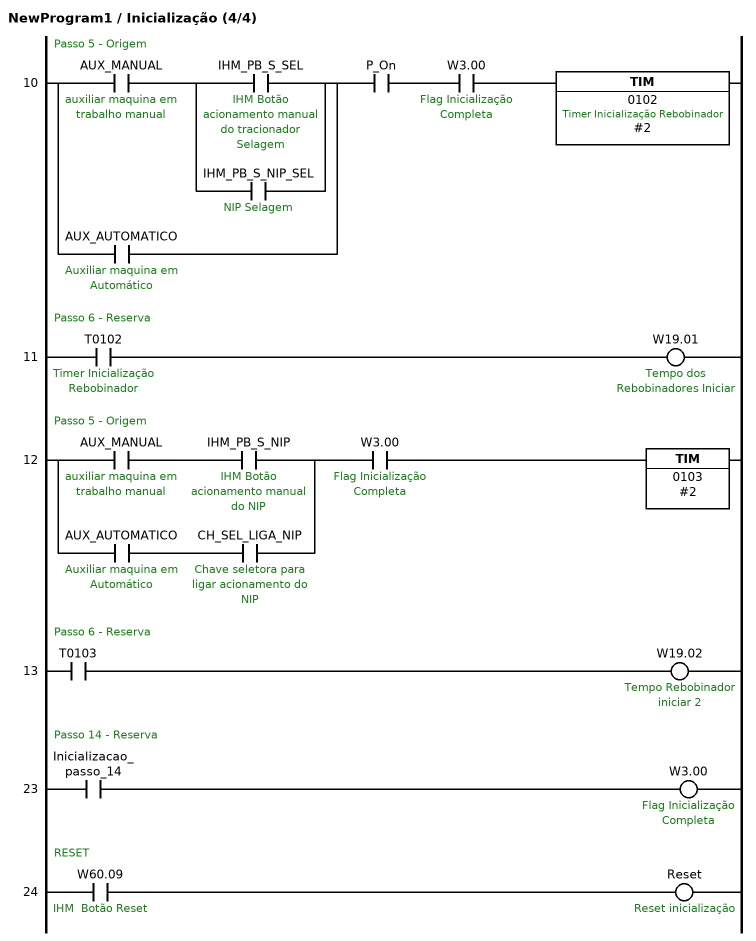
; [picture p24: NewProgram1 / Inicialização, rungs 10-24]
; rung 10: Passo 5 - Origem
LD AUX_MANUAL  ; auxiliar maquina em trabalho manual
LD IHM_PB_S_SEL  ; IHM Botão acionamento manual do tracionador Selagem
OR IHM_PB_S_NIP_SEL  ; NIP Selagem
ANDLD
OR AUX_AUTOMATICO  ; Auxiliar maquina em Automático
AND P_On
AND W3.00  ; Flag Inicialização Completa
TIM 0102 #2  ; Timer Inicialização Rebobinador
; rung 11: Passo 6 - Reserva
LD T0102  ; Timer Inicialização Rebobinador
OUT W19.01  ; Tempo dos Rebobinadores Iniciar
; rung 12: Passo 5 - Origem
LD AUX_MANUAL  ; auxiliar maquina em trabalho manual
AND IHM_PB_S_NIP  ; IHM Botão acionamento manual do NIP
LD AUX_AUTOMATICO  ; Auxiliar maquina em Automático
AND CH_SEL_LIGA_NIP  ; Chave seletora para ligar acionamento do NIP
ORLD
AND W3.00  ; Flag Inicialização Completa
TIM 0103 #2
; rung 13: Passo 6 - Reserva
LD T0103
OUT W19.02  ; Tempo Rebobinador iniciar 2
; rung 14: Passo 5 - Origem
; rung 15: Passo 6 - Reserva
; rung 16: Passo 7 - Reserva
; rung 17: Passo 8 - Reserva
; rung 18: Passo 9 - Reserva
; rung 19: Passo 10 - Reserva
; rung 20: Passo 11 - Reserva
; rung 21: Passo 12 - Reserva
; rung 22: Passo 13 - Reserva
; rung 23: Passo 14 - Reserva
LD Inicializacao_passo_14
OUT W3.00  ; Flag Inicialização Completa
; rung 24: RESET
LD W60.09  ; IHM  Botão Reset
OUT Reset  ; Reset inicialização

### Section Temperatura

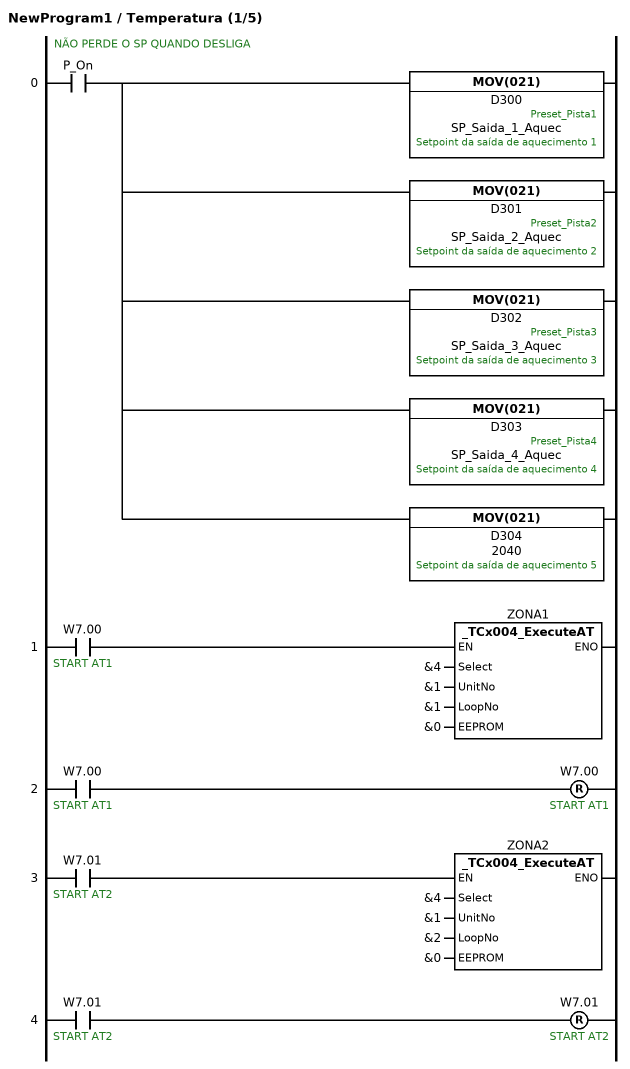
; rung 0: NÃO PERDE O SP QUANDO DESLIGA
LD P_On
MOV(021) D300 SP_Saida_1_Aquec  ; Preset_Pista1, Setpoint da saída de aquecimento 1
MOV(021) D301 SP_Saida_2_Aquec  ; Preset_Pista2, Setpoint da saída de aquecimento 2
MOV(021) D302 SP_Saida_3_Aquec  ; Preset_Pista3, Setpoint da saída de aquecimento 3
MOV(021) D303 SP_Saida_4_Aquec  ; Preset_Pista4, Setpoint da saída de aquecimento 4
MOV(021) D304 2040  ; Setpoint da saída de aquecimento 5
; rung 1
LD W7.00  ; START AT1
CALL ZONA1 : _TCx004_ExecuteAT (Select := &4, UnitNo := &1, LoopNo := &1, EEPROM := &0)
; rung 2
LD W7.00  ; START AT1
RSET W7.00  ; START AT1
; rung 3
LD W7.01  ; START AT2
CALL ZONA2 : _TCx004_ExecuteAT (Select := &4, UnitNo := &1, LoopNo := &2, EEPROM := &0)
; rung 4
LD W7.01  ; START AT2
RSET W7.01  ; START AT2

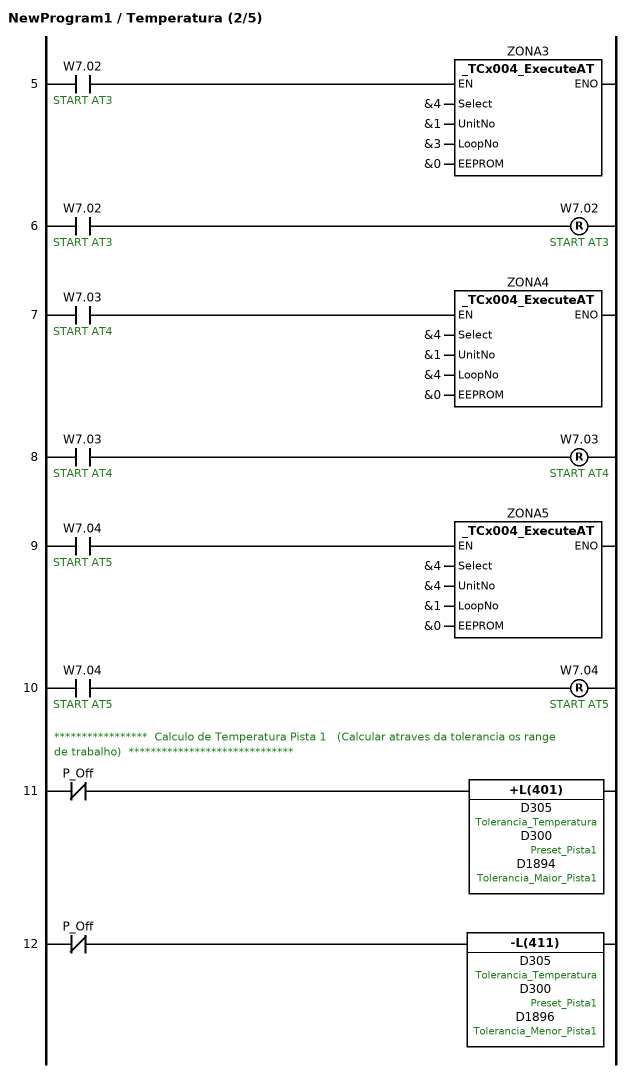
; rung 5
LD W7.02  ; START AT3
CALL ZONA3 : _TCx004_ExecuteAT (Select := &4, UnitNo := &1, LoopNo := &3, EEPROM := &0)
; rung 6
LD W7.02  ; START AT3
RSET W7.02  ; START AT3
; rung 7
LD W7.03  ; START AT4
CALL ZONA4 : _TCx004_ExecuteAT (Select := &4, UnitNo := &1, LoopNo := &4, EEPROM := &0)
; rung 8
LD W7.03  ; START AT4
RSET W7.03  ; START AT4
; rung 9
LD W7.04  ; START AT5
CALL ZONA5 : _TCx004_ExecuteAT (Select := &4, UnitNo := &4, LoopNo := &1, EEPROM := &0)
; rung 10
LD W7.04  ; START AT5
RSET W7.04  ; START AT5
; rung 11: *****************  Calculo de Temperatura Pista 1   (Calcular atraves da tolerancia os range de trabalho)  ******************************
LDNOT P_Off
+L(401) D305 D300 D1894  ; Tolerancia_Temperatura, Preset_Pista1, Tolerancia_Maior_Pista1
; rung 12
LDNOT P_Off
-L(411) D305 D300 D1896  ; Tolerancia_Temperatura, Preset_Pista1, Tolerancia_Menor_Pista1

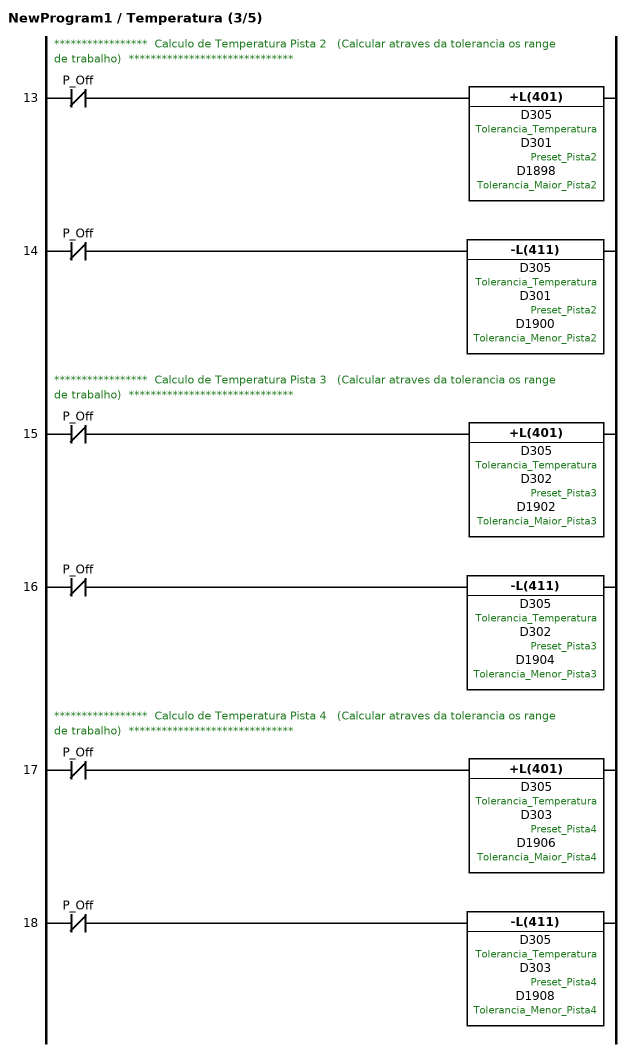
; rung 13: *****************  Calculo de Temperatura Pista 2   (Calcular atraves da tolerancia os range de trabalho)  ******************************
LDNOT P_Off
+L(401) D305 D301 D1898  ; Tolerancia_Temperatura, Preset_Pista2, Tolerancia_Maior_Pista2
; rung 14
LDNOT P_Off
-L(411) D305 D301 D1900  ; Tolerancia_Temperatura, Preset_Pista2, Tolerancia_Menor_Pista2
; rung 15: *****************  Calculo de Temperatura Pista 3   (Calcular atraves da tolerancia os range de trabalho)  ******************************
LDNOT P_Off
+L(401) D305 D302 D1902  ; Tolerancia_Temperatura, Preset_Pista3, Tolerancia_Maior_Pista3
; rung 16
LDNOT P_Off
-L(411) D305 D302 D1904  ; Tolerancia_Temperatura, Preset_Pista3, Tolerancia_Menor_Pista3
; rung 17: *****************  Calculo de Temperatura Pista 4   (Calcular atraves da tolerancia os range de trabalho)  ******************************
LDNOT P_Off
+L(401) D305 D303 D1906  ; Tolerancia_Temperatura, Preset_Pista4, Tolerancia_Maior_Pista4
; rung 18
LDNOT P_Off
-L(411) D305 D303 D1908  ; Tolerancia_Temperatura, Preset_Pista4, Tolerancia_Menor_Pista4

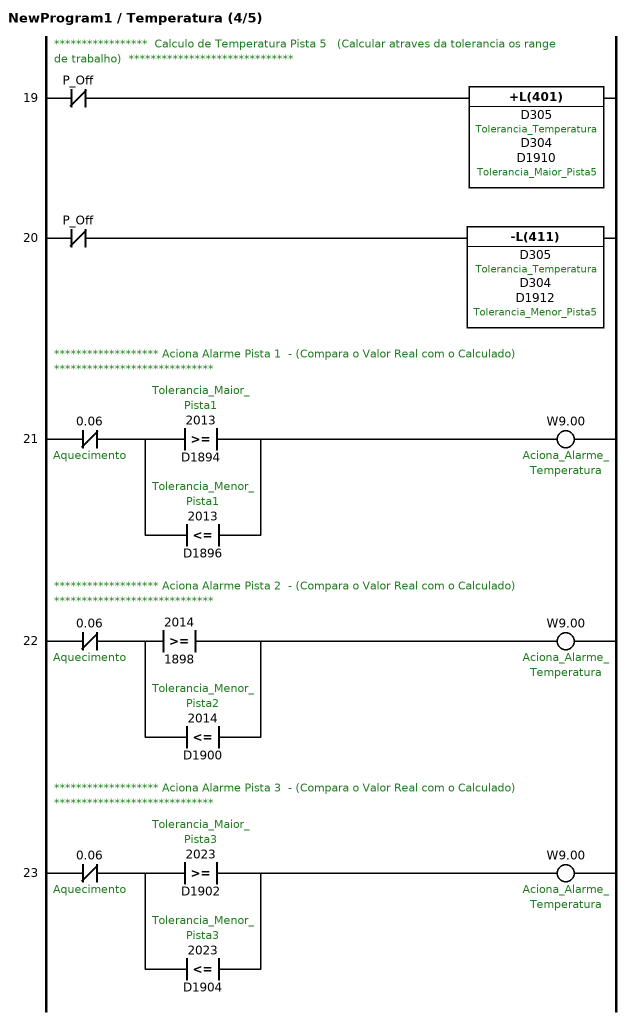
; rung 19: *****************  Calculo de Temperatura Pista 5   (Calcular atraves da tolerancia os range de trabalho)  ******************************
LDNOT P_Off
+L(401) D305 D304 D1910  ; Tolerancia_Temperatura, Tolerancia_Maior_Pista5
; rung 20
LDNOT P_Off
-L(411) D305 D304 D1912  ; Tolerancia_Temperatura, Tolerancia_Menor_Pista5
; rung 21: ******************* Aciona Alarme Pista 1  - (Compara o Valor Real com o Calculado) *****************************
LDNOT 0.06  ; Aquecimento
LD>=L(326) 2013 D1894  ; Tolerancia_Maior_Pista1
OR<=L(316) 2013 D1896  ; Tolerancia_Menor_Pista1
ANDLD
OUT W9.00  ; Aciona_Alarme_Temperatura
; rung 22: ******************* Aciona Alarme Pista 2  - (Compara o Valor Real com o Calculado) *****************************
LDNOT 0.06  ; Aquecimento
LD>=L(326) 2014 1898
OR<=L(316) 2014 D1900  ; Tolerancia_Menor_Pista2
ANDLD
OUT W9.00  ; Aciona_Alarme_Temperatura
; rung 23: ******************* Aciona Alarme Pista 3  - (Compara o Valor Real com o Calculado) *****************************
LDNOT 0.06  ; Aquecimento
LD>=L(326) 2023 D1902  ; Tolerancia_Maior_Pista3
OR<=L(316) 2023 D1904  ; Tolerancia_Menor_Pista3
ANDLD
OUT W9.00  ; Aciona_Alarme_Temperatura

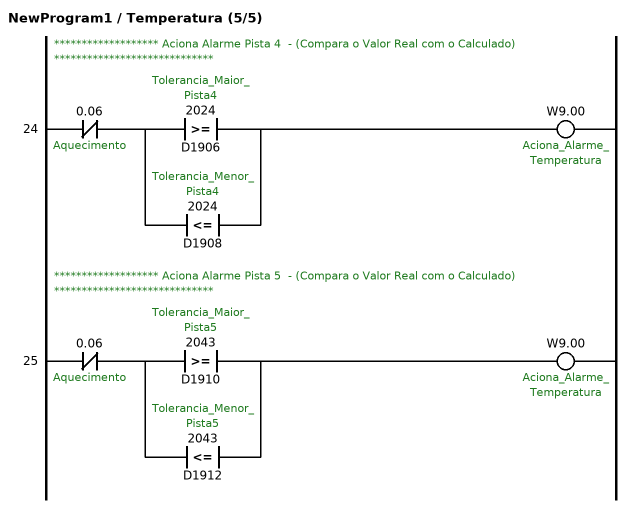
; rung 24: ******************* Aciona Alarme Pista 4  - (Compara o Valor Real com o Calculado) *****************************
LDNOT 0.06  ; Aquecimento
LD>=L(326) 2024 D1906  ; Tolerancia_Maior_Pista4
OR<=L(316) 2024 D1908  ; Tolerancia_Menor_Pista4
ANDLD
OUT W9.00  ; Aciona_Alarme_Temperatura
; rung 25: ******************* Aciona Alarme Pista 5  - (Compara o Valor Real com o Calculado) *****************************
LDNOT 0.06  ; Aquecimento
LD>=L(326) 2043 D1910  ; Tolerancia_Maior_Pista5
OR<=L(316) 2043 D1912  ; Tolerancia_Menor_Pista5
ANDLD
OUT W9.00  ; Aciona_Alarme_Temperatura

### Section Automático

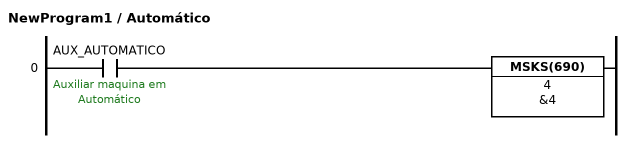
; rung 0
LD AUX_AUTOMATICO  ; Auxiliar maquina em Automático
MSKS(690) 4 &4

### Section Producao

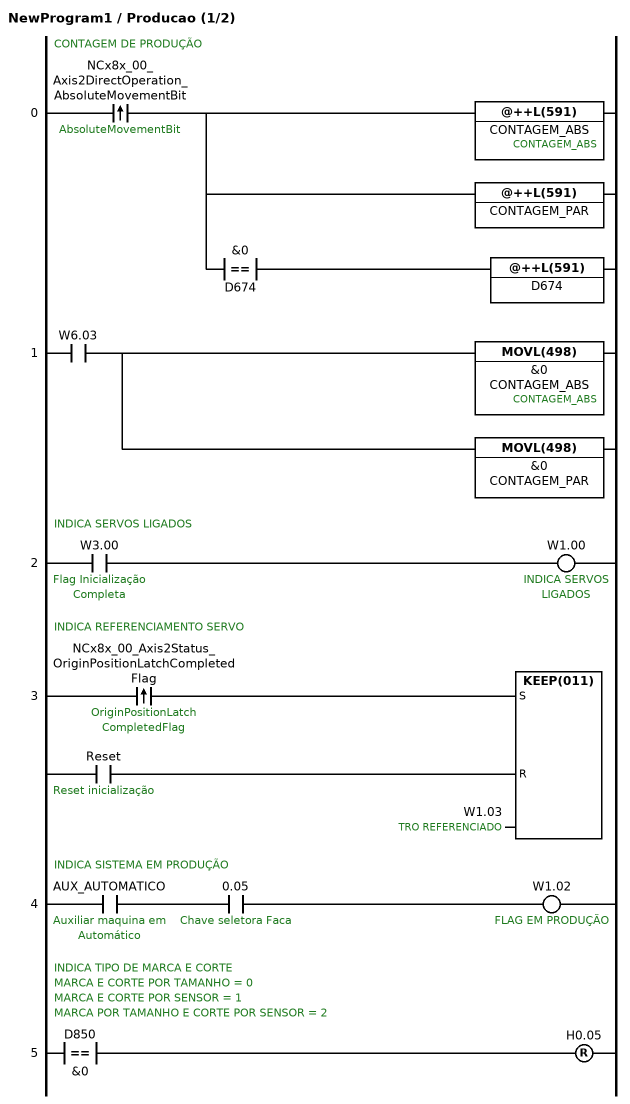
; rung 0: CONTAGEM DE PRODUÇÃO
@LD NCx8x_00_Axis2DirectOperation_AbsoluteMovementBit  ; AbsoluteMovementBit
@++L(591) CONTAGEM_ABS  ; CONTAGEM_ABS
@++L(591) CONTAGEM_PAR
AND=(300) &0 D674
@++L(591) D674
; rung 1
LD W6.03
MOVL(498) &0 CONTAGEM_ABS  ; CONTAGEM_ABS
MOVL(498) &0 CONTAGEM_PAR
; rung 2: INDICA SERVOS LIGADOS
LD W3.00  ; Flag Inicialização Completa
OUT W1.00  ; INDICA SERVOS LIGADOS
; rung 3: INDICA REFERENCIAMENTO SERVO
@LD NCx8x_00_Axis2Status_OriginPositionLatchCompletedFlag  ; OriginPositionLatchCompletedFlag
LD Reset  ; Reset inicialização
KEEP(011) W1.03  ; TRO REFERENCIADO
; rung 4: INDICA SISTEMA EM PRODUÇÃO
LD AUX_AUTOMATICO  ; Auxiliar maquina em Automático
AND 0.05  ; Chave seletora Faca
OUT W1.02  ; FLAG EM PRODUÇÃO
; rung 5: INDICA TIPO DE MARCA E CORTE / MARCA E CORTE POR TAMANHO = 0 / MARCA E CORTE POR SENSOR = 1 / MARCA POR TAMANHO E CORTE POR SENSOR = 2
LD=(300) D850 &0
RSET H0.05

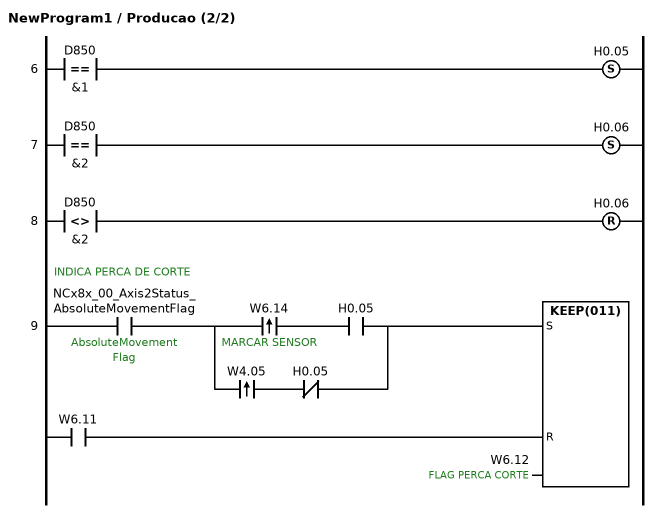
; rung 6
LD=(300) D850 &1
SET H0.05
; rung 7
LD=(300) D850 &2
SET H0.06
; rung 8
LD<>(305) D850 &2
RSET H0.06
; rung 9: INDICA PERCA DE CORTE
LD NCx8x_00_Axis2Status_AbsoluteMovementFlag  ; AbsoluteMovementFlag
@LD W6.14  ; MARCAR SENSOR
AND H0.05
@LD W4.05
ANDNOT H0.05
ORLD
ANDLD
LD W6.11
KEEP(011) W6.12  ; FLAG PERCA CORTE

### Section Sensor

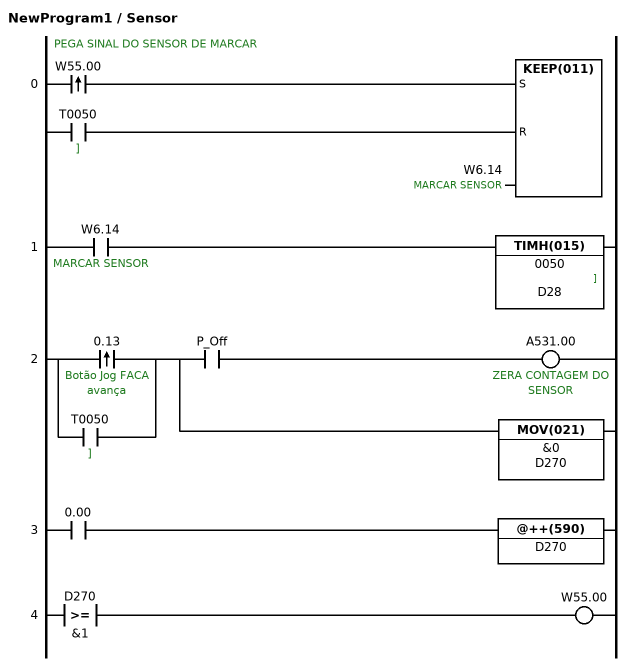
; rung 0: PEGA SINAL DO SENSOR DE MARCAR
@LD W55.00
LD T0050  ; ]
KEEP(011) W6.14  ; MARCAR SENSOR
; rung 1
LD W6.14  ; MARCAR SENSOR
TIMH(015) 0050 D28  ; ]
; rung 2
@LD 0.13  ; Botão Jog FACA avança
OR T0050  ; ]
OUT TR0
AND P_Off
OUT A531.00  ; ZERA CONTAGEM DO SENSOR
LD TR0
MOV(021) &0 D270
; rung 3
LD 0.00
@++(590) D270
; rung 4
LD>=(325) D270 &1
OUT W55.00

### Section Etiquetador

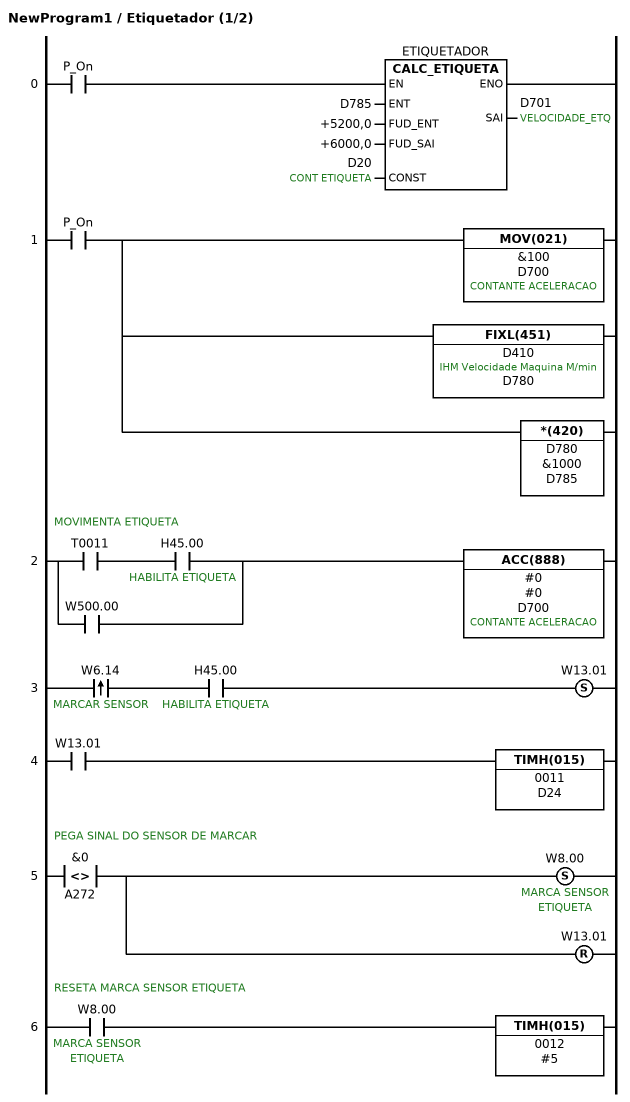
; rung 0
LD P_On
CALL ETIQUETADOR : CALC_ETIQUETA (ENT := D785, FUD_ENT := +5200,0, FUD_SAI := +6000,0, CONST := D20, SAI => D701)  ; CONT ETIQUETA, VELOCIDADE_ETQ
; rung 1
LD P_On
MOV(021) &100 D700  ; CONTANTE ACELERACAO
FIXL(451) D410 D780  ; IHM Velocidade Maquina M/min
*(420) D780 &1000 D785
; rung 2: MOVIMENTA ETIQUETA
LD T0011
AND H45.00  ; HABILITA ETIQUETA
OR W500.00
ACC(888) #0 #0 D700  ; CONTANTE ACELERACAO
; rung 3
@LD W6.14  ; MARCAR SENSOR
AND H45.00  ; HABILITA ETIQUETA
SET W13.01
; rung 4
LD W13.01
TIMH(015) 0011 D24
; rung 5: PEGA SINAL DO SENSOR DE MARCAR
LD<>(305) &0 A272
SET W8.00  ; MARCA SENSOR ETIQUETA
RSET W13.01
; rung 6: RESETA MARCA SENSOR ETIQUETA
LD W8.00  ; MARCA SENSOR ETIQUETA
TIMH(015) 0012 #5

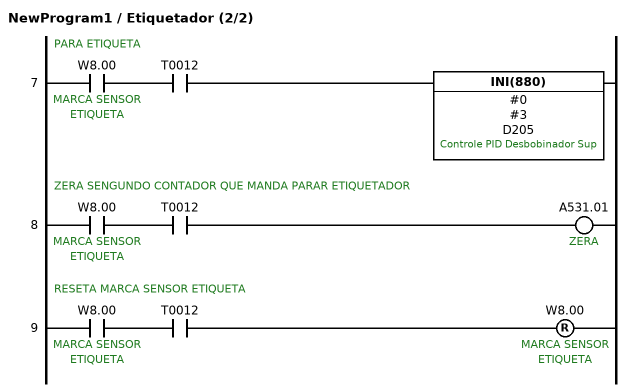
; rung 7: PARA ETIQUETA
LD W8.00  ; MARCA SENSOR ETIQUETA
AND T0012
INI(880) #0 #3 D205  ; Controle PID Desbobinador Sup
; rung 8: ZERA SENGUNDO CONTADOR QUE MANDA PARAR ETIQUETADOR
LD W8.00  ; MARCA SENSOR ETIQUETA
AND T0012
OUT A531.01  ; ZERA
; rung 9: RESETA MARCA SENSOR ETIQUETA
LD W8.00  ; MARCA SENSOR ETIQUETA
AND T0012
RSET W8.00  ; MARCA SENSOR ETIQUETA

### Section Receita

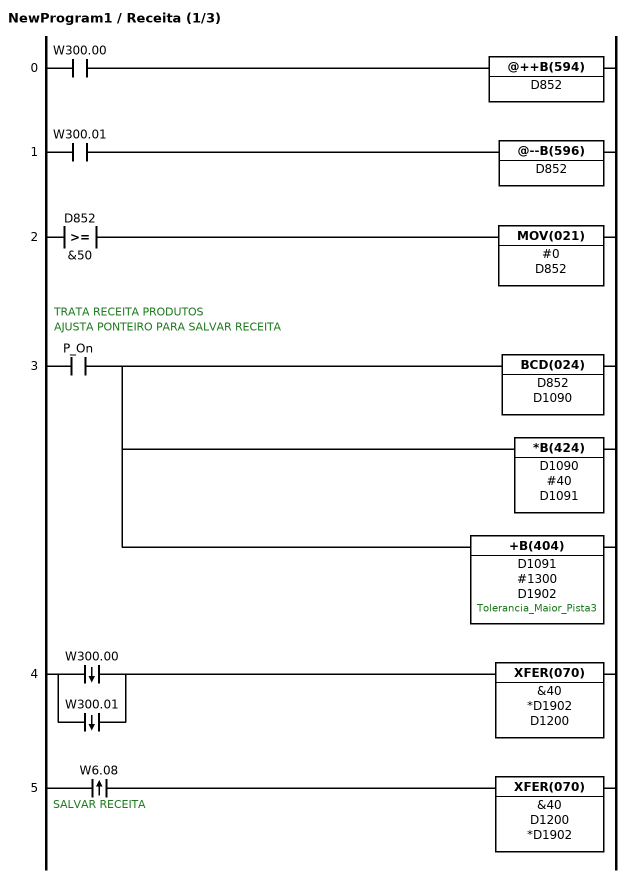
; rung 0
LD W300.00
@++B(594) D852
; rung 1
LD W300.01
@--B(596) D852
; rung 2
LD>=(325) D852 &50
MOV(021) #0 D852
; rung 3: TRATA RECEITA PRODUTOS / AJUSTA PONTEIRO PARA SALVAR RECEITA
LD P_On
BCD(024) D852 D1090
*B(424) D1090 #40 D1091
+B(404) D1091 #1300 D1902  ; Tolerancia_Maior_Pista3
; rung 4
%LD W300.00
%OR W300.01
XFER(070) &40 *D1902 D1200
; rung 5
@LD W6.08  ; SALVAR RECEITA
XFER(070) &40 D1200 *D1902

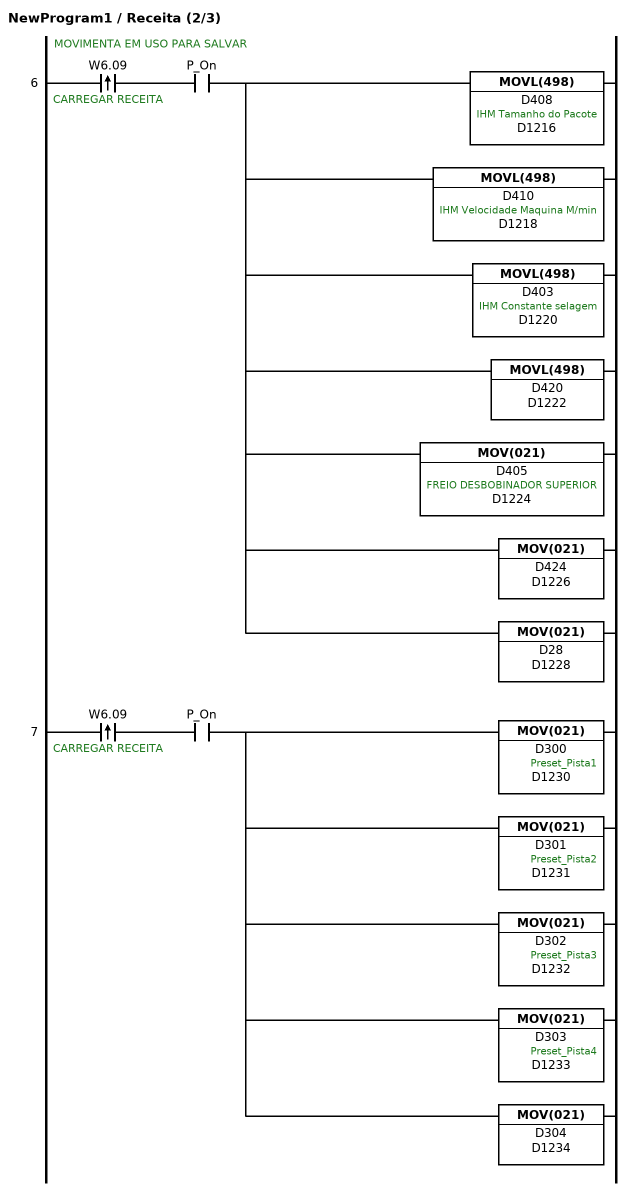
; rung 6: MOVIMENTA EM USO PARA SALVAR
@LD W6.09  ; CARREGAR RECEITA
AND P_On
MOVL(498) D408 D1216  ; IHM Tamanho do Pacote
MOVL(498) D410 D1218  ; IHM Velocidade Maquina M/min
MOVL(498) D403 D1220  ; IHM Constante selagem
MOVL(498) D420 D1222
MOV(021) D405 D1224  ; FREIO DESBOBINADOR SUPERIOR
MOV(021) D424 D1226
MOV(021) D28 D1228
; rung 7
@LD W6.09  ; CARREGAR RECEITA
AND P_On
MOV(021) D300 D1230  ; Preset_Pista1
MOV(021) D301 D1231  ; Preset_Pista2
MOV(021) D302 D1232  ; Preset_Pista3
MOV(021) D303 D1233  ; Preset_Pista4
MOV(021) D304 D1234

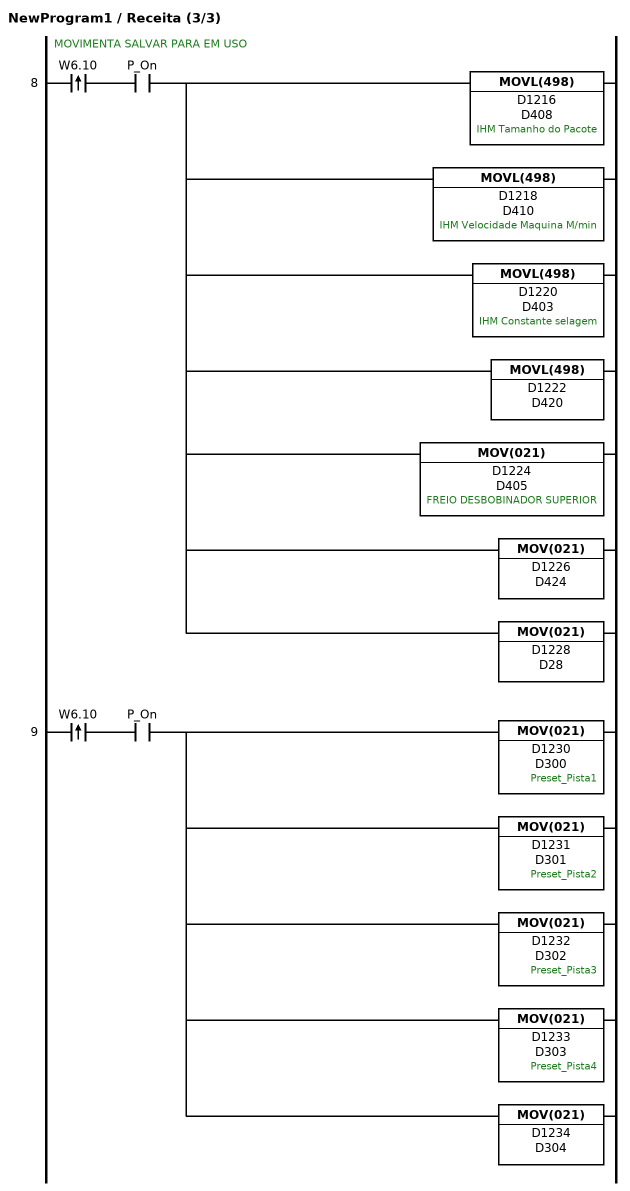
; rung 8: MOVIMENTA SALVAR PARA EM USO
@LD W6.10
AND P_On
MOVL(498) D1216 D408  ; IHM Tamanho do Pacote
MOVL(498) D1218 D410  ; IHM Velocidade Maquina M/min
MOVL(498) D1220 D403  ; IHM Constante selagem
MOVL(498) D1222 D420
MOV(021) D1224 D405  ; FREIO DESBOBINADOR SUPERIOR
MOV(021) D1226 D424
MOV(021) D1228 D28
; rung 9
@LD W6.10
AND P_On
MOV(021) D1230 D300  ; Preset_Pista1
MOV(021) D1231 D301  ; Preset_Pista2
MOV(021) D1232 D302  ; Preset_Pista3
MOV(021) D1233 D303  ; Preset_Pista4
MOV(021) D1234 D304

### Section END
; rung 0
END(001)

## Program Comparação_pacote (interrupt task 2)

### Section Section1

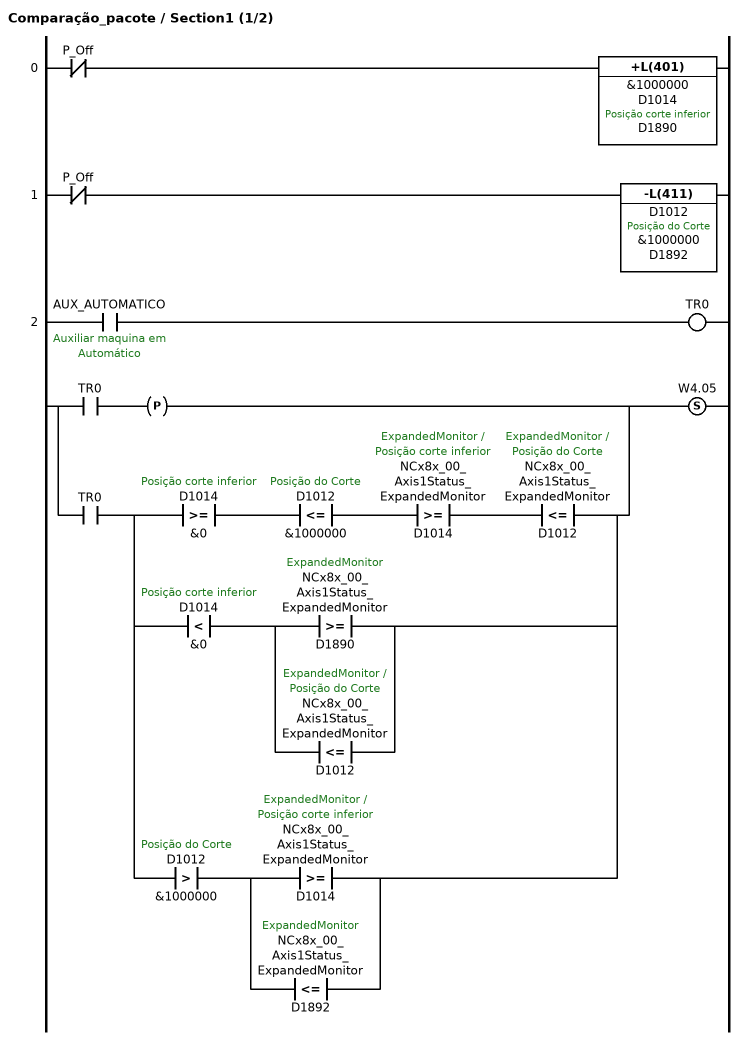
; rung 0
LDNOT P_Off
+L(401) &1000000 D1014 D1890  ; Posição corte inferior
; rung 1
LDNOT P_Off
-L(411) D1012 &1000000 D1892  ; Posição do Corte
; rung 2
LD AUX_AUTOMATICO  ; Auxiliar maquina em Automático
OUT TR0
UP(521)
LD TR0
LD>=L(326) D1014 &0  ; Posição corte inferior
AND<=L(316) D1012 &1000000  ; Posição do Corte
AND>=L(326) NCx8x_00_Axis1Status_ExpandedMonitor D1014  ; ExpandedMonitor, Posição corte inferior
AND<=L(316) NCx8x_00_Axis1Status_ExpandedMonitor D1012  ; ExpandedMonitor, Posição do Corte
LD<SL(313) D1014 &0  ; Posição corte inferior
LD>=L(326) NCx8x_00_Axis1Status_ExpandedMonitor D1890  ; ExpandedMonitor
OR<=L(316) NCx8x_00_Axis1Status_ExpandedMonitor D1012  ; ExpandedMonitor, Posição do Corte
ANDLD
ORLD
LD>L(321) D1012 &1000000  ; Posição do Corte
LD>=L(326) NCx8x_00_Axis1Status_ExpandedMonitor D1014  ; ExpandedMonitor, Posição corte inferior
OR<=L(316) NCx8x_00_Axis1Status_ExpandedMonitor D1892  ; ExpandedMonitor
ANDLD
ORLD
ANDLD
ORLD
SET W4.05

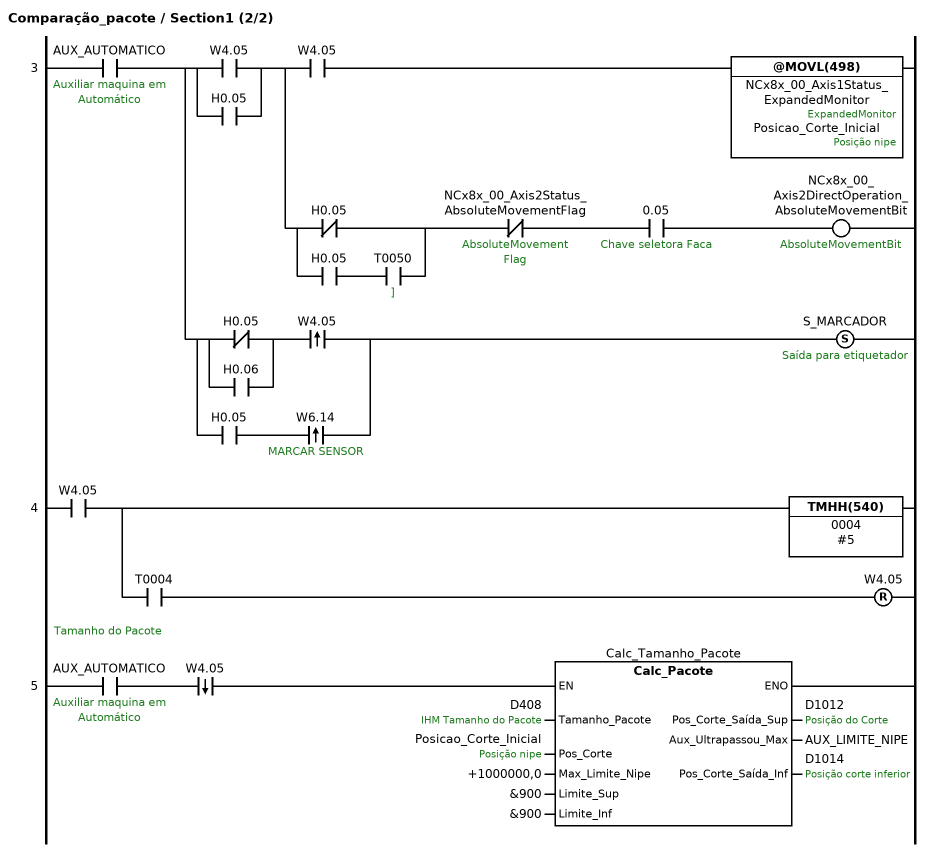
; rung 3
LD AUX_AUTOMATICO  ; Auxiliar maquina em Automático
OUT TR0
LD W4.05
OR H0.05
ANDLD
OUT TR1
AND W4.05
@MOVL(498) NCx8x_00_Axis1Status_ExpandedMonitor Posicao_Corte_Inicial  ; ExpandedMonitor, Posição nipe
LD TR1
LDNOT H0.05
LD H0.05
AND T0050  ; ]
ORLD
ANDLD
ANDNOT NCx8x_00_Axis2Status_AbsoluteMovementFlag  ; AbsoluteMovementFlag
AND 0.05  ; Chave seletora Faca
OUT NCx8x_00_Axis2DirectOperation_AbsoluteMovementBit  ; AbsoluteMovementBit
LD TR0
LDNOT H0.05
OR H0.06
@AND W4.05
LD H0.05
@AND W6.14  ; MARCAR SENSOR
ORLD
ANDLD
SET S_MARCADOR  ; Saída para etiquetador
; rung 4
LD W4.05
TMHH(540) 0004 #5
AND T0004
RSET W4.05
; rung 5: Tamanho do Pacote
LD AUX_AUTOMATICO  ; Auxiliar maquina em Automático
%AND W4.05
CALL Calc_Tamanho_Pacote : Calc_Pacote (Tamanho_Pacote := D408, Pos_Corte := Posicao_Corte_Inicial, Max_Limite_Nipe := +1000000,0, Limite_Sup := &900, Limite_Inf := &900, Pos_Corte_Saída_Sup => D1012, Aux_Ultrapassou_Max => AUX_LIMITE_NIPE, Pos_Corte_Saída_Inf => D1014)  ; IHM Tamanho do Pacote, Posição nipe, Posição do Corte, Posição corte inferior

### Section END
; rung 0
END(001)

## Function block _TCx004_ExecuteAT (Omron library block, body left out)

## Function block CALC_ETIQUETA
VAR_INPUT
  ENT : INT;
  FUD_ENT : LREAL;
  FUD_SAI : LREAL;
  CONST : INT;
END_VAR
VAR_OUTPUT
  SAI : DINT;
END_VAR
VAR
  ENT1 : LREAL;
  SAI1 : LREAL;
  CONST1 : LREAL;
END_VAR
ENT1 := INT_TO_LREAL(ENT);
CONST1 := INT_TO_LREAL(CONST);
CONST1 := CONST1/10000,0;
SAI1 := (ENT1*FUD_SAI)/FUD_ENT;
SAI1:= SAI1*CONST1;
SAI  := LREAL_TO_DINT (SAI1);

## Function block Calc_Pacote
VAR_INPUT
  Tamanho_Pacote : REAL;
  Pos_Corte : DINT;
  Max_Limite_Nipe : REAL;
  Limite_Sup : DINT;
  Limite_Inf : DINT;
END_VAR
VAR_OUTPUT
  Pos_Corte_Saída_Sup : DINT;
  Aux_Ultrapassou_Max : BOOL;
  Pos_Corte_Saída_Inf : DINT;
END_VAR
VAR
  pacote_mm : REAL;
  pos_corte_real : REAL;
END_VAR
pos_corte_real:= DINT_TO_REAL(Pos_Corte);
pacote_mm:= (Tamanho_Pacote*+1000,00)+pos_corte_real;
IF pacote_mm <Max_Limite_Nipe THEN
	Pos_Corte_Saída_Sup:= (REAL_TO_DINT(pacote_mm))+Limite_Sup;
	Pos_Corte_Saída_Inf:=  (REAL_TO_DINT(pacote_mm))-Limite_Inf;
	Aux_Ultrapassou_Max:= FALSE;
ELSE
	Pos_Corte_Saída_Sup:=(REAL_TO_DINT(pacote_mm-Max_Limite_Nipe))+Limite_Sup;
	Pos_Corte_Saída_Inf:= (REAL_TO_DINT(pacote_mm-Max_Limite_Nipe))-Limite_Inf;
	Aux_Ultrapassou_Max:= TRUE;
END_IF;

## Function block Calc_Vel
VAR_INPUT
  Vel_Maq : REAL;
  K_Constante : REAL;  (* Constante de velocidade 0 a 200% *)
END_VAR
VAR_OUTPUT
  Vel_Servo : DINT;
END_VAR
VAR
  k_fator_mult : REAL;
  vel_fator : REAL;
END_VAR
k_fator_mult:= K_Constante/+100,00;
vel_fator:= ((Vel_Maq/+60,00)*+1000,00)*+1000,00*k_fator_mult;
Vel_Servo:= REAL_TO_DINT(vel_fator);

## Function block Calc_Vel_TRO
VAR_INPUT
  K_Constante : REAL;
  Vel_Maq : REAL;
END_VAR
VAR_OUTPUT
  Vel_Servo : DINT;
END_VAR
VAR
  k_fator_mult : REAL;
  vel_fator : REAL;
END_VAR
k_fator_mult:= K_Constante/+100,00;
vel_fator:= (((Vel_Maq*+8,33394722)/+60,00)*+1000,00)*+1000,00*k_fator_mult;
Vel_Servo:= REAL_TO_DINT(vel_fator);

## Function block Escala_SA
VAR_INPUT
  Entrada : REAL;
  Max_Entrada : REAL;
  Resolucao_SA : REAL;
END_VAR
VAR_OUTPUT
  Saida_Escala : INT;
END_VAR
VAR
  aux_sa : REAL;
  fator_multi : REAL;
END_VAR
fator_multi:= (Max_Entrada/Resolucao_SA);
aux_sa:= Entrada/fator_multi;
Saida_Escala:=REAL_TO_INT(aux_sa);

## Function block Relacao_motor
VAR_INPUT
  Pos_Des : LREAL;
  Reducao : LREAL;
  Rot_Servo_Motor : LREAL;
  Distancia_max : LREAL;
END_VAR
VAR_OUTPUT
  Saida_Vel : DINT;
  Saida_Pos : DINT;
END_VAR
VAR
  aux_saida_pos_real : LREAL;
  aux_saida_vel_real : LREAL;
END_VAR
aux_saida_vel_real:= Rot_Servo_Motor/Reducao;
aux_saida_pos_real:= Pos_Des*Reducao;
Saida_Pos:= LREAL_TO_DINT(aux_saida_pos_real); 
Saida_Vel:= LREAL_TO_DINT(aux_saida_vel_real);